// TIA Portal project "vfd-spindel-plc_v20" (V20)

(* hardware
DEVICE "ET 200SP station_1"  ET 200SP-Station
   slot 0: "Rack_0"  Rack  6ES5 710-8MAx1
   slot 1: "vfd-spindel-plc"  CPU 1510SP-1 PN  6ES7 510-1DJ01-0AB0  V2.5
      slot 32768: "PROFINET interface_1"  X1
         slot 32771: "Port_3"  X1 P3
   slot 2: "AQ 4xU/I ST_1"  AQ 4xU/I ST  6ES7 135-6HD00-0BA1  V1.1
      slot 1: "AQ 4xU/I ST_1"  AQ 4xU/I ST
   slot 3: "AI 2xU/I 2-/4-wire HS_1"  AI 2xU/I 2-,4-wire HS  6ES7 134-6HB00-0DA1  V2.0
      slot 1: "AI 2xU/I 2-/4-wire HS_1"  AI 2xU/I 2-,4-wire HS
   slot 4: "DQ 8x24VDC/0.5A HF_1"  DQ 8x24VDC/0.5A HF  6ES7 132-6BF00-0CA0  V2.0
      slot 1: "DQ 8x24VDC/0.5A HF_1"  DQ 8x24VDC/0.5A HF
   slot 5: "DQ 8x24VDC/0.5A HF_2"  DQ 8x24VDC/0.5A HF  6ES7 132-6BF00-0CA0  V2.0
      slot 1: "DQ 8x24VDC/0.5A HF_2"  DQ 8x24VDC/0.5A HF
   slot 6: "DI 8x24VDC HF_1"  DI 8x24VDC HF  6ES7 131-6BF00-0CA0  V2.0
      slot 1: "DI 8x24VDC HF_1"  DI 8x24VDC HF
   slot 7: "TM Count 1x24V_1"  TM Count 1x24V  6ES7 138-6AA01-0BA0  V2.0
      slot 1: "TM Count 1x24V_1"  TM Count 1x24V
   slot 8: "AI 4xRTD/TC 2-/3-/4-wire HF_1"  AI 4xRTD/TC 2-,3-,4-wire HF  6ES7 134-6JD00-0CA1  V2.0
      slot 1: "AI 4xRTD/TC 2-/3-/4-wire HF_1"  AI 4xRTD/TC 2-,3-,4-wire HF
   slot 9: "Server module_1"  Server module  6ES7 193-6PA00-0AA0  V1.1
      slot 1: "Server module_1"  Server module
   slot 127: "BA 2xRJ45"  BA 2xRJ45  6ES7 193-6AR00-0AA0  V0.0
      slot 32769: "Port_1"  X1 P1  6ES7 193-6AR00-0AA0
      slot 32770: "Port_2"  X1 P2  6ES7 193-6AR00-0AA0
DEVICE "ktp700_basic"  KTP700 Basic PN
   slot 0: "ktp700_basic"  KTP700 Basic PN  6AV2 123-2GB03-0AX0  17.0.0.0
   slot 1: "HMI_RT_1"  KTP700 Basic PN  6AV2 123-2GB03-0AX0  17.0.0.0
   slot 5: "ktp700_basic.IE_CP_1"  PROFINET Interface  17.0.0.0
      slot 1: "PROFINET Interface_1"  PROFINET Interface
         slot 1: "Port_1"  Port
*)

// ===== PLC "vfd-spindel-plc"  CPU 1510SP-1 PN =====

VAR_GLOBAL   // PLC tag table "Default tag table"
   "DQ0" AT %Q8.0 : Bool;
   "AQ_Ch1" AT %QW0 : Word;
   "AI_Ch0" AT %IW0 : Word;
   "AQ_Ch2" AT %QW2 : Word;
   "AI_Ch1" AT %IW2 : Word;
   "AQ_Ch3" AT %QW4 : Word;
   "AQ_Ch4" AT %QW6 : Word;
   "DI4" AT %I28.3 : Bool;   // Safety relay
   "DI5" AT %I28.4 : Bool;   // Safety button
   "AI1_RTD" AT %IW6 : Word;
   "AI2_RTD" AT %IW8 : Word;
   "DI0_safetyRelay" AT %I28.0 : Bool;
   "DQ1" AT %Q8.1 : Bool;
   "DQ4" AT %Q8.4 : Bool;
   "DI1_SafetyRelay_State" AT %I28.1 : Bool;
END_VAR

TYPE "UDT_IO_AI"
   STRUCT
      AI1_TeplotaKomaraKartac_Ohm : Int;
   END_STRUCT;
END_TYPE

TYPE "UDT_IO_AQ"
   STRUCT
      SpeedVoltage : Real;
      AQ2_VoltageCtrl_V : Real;
      AQ3_CurrentCtrl_V : Real;
   END_STRUCT;
END_TYPE

TYPE "UDT_IO_DI"
   STRUCT
      SafetyRelayAuxOk : Bool;
      HSC_Couter : UInt;
      EmergencyStop : Bool;
      ExternalFault : Bool;
   END_STRUCT;
END_TYPE

TYPE "UDT_IO_DQ"
   STRUCT
      EmergencyStop : Bool;
      RunForwardCmd : Bool;
      FaultResetCmd : Bool;
      MultiSpeed1 : Bool;
      ExternalFault : Bool;
      DO_OutputOff : Bool;
   END_STRUCT;
END_TYPE

TYPE "UDT_LABPSU_STATUS"
   STRUCT
      VoltageSet_V : Real;
      CurrentSet_A : Real;
      State : USInt;
      StatusText : String[40];
   END_STRUCT;
END_TYPE

TYPE "UDT_SPINDEL_STATUS"
   STRUCT
      RunLatched : Bool;
      TripActive : Bool;
      State : USInt;
      StatusText : String[40];
   END_STRUCT;
END_TYPE

TYPE "UDT_SAFETY_STATUS"
   STRUCT
      SafetyOk : Bool;
      PermitMotion : Bool;
      TripActive : Bool;
      TripCode : USInt;
      StatusText : String[40];
   END_STRUCT;
END_TYPE

DATA_BLOCK "DAC"   // DB2
{ S7_Optimized_Access := 'TRUE' }
VERSION : 0.1
   VAR
      IccLimiter : Struct
         MaxOutputCurrent : Int := 60;
         MinOutputCurrent : Int := 0;
         MinDacRange : Int := 0;
         MaxDacRange : Int := 27648;
         value : UInt := 0;
      END_STRUCT;
      UccVoltage : Struct
         MaxOutput : Int := 10;
         MinOutput : Int := 0;
         MinDacRange : Int := 0;
         MaxDacRange : Int := 27648;
      END_STRUCT;
      VFD : Struct
         MaxFrequency : Int := 18000;
         MinFrequency : Int := 0;
         MinDacRange : Int := 0;
         value : UInt := 0;
         MaxDacRange : Int := 27648;
      END_STRUCT;
      Sinus : Struct
         Value : Real := 0.0;
         Sample : Int := 0;
         Amplitude : Real := 1.0;
         Period : Real := 1.0;
         SamplePeriod : Real := 0.01;
      END_STRUCT;
   END_VAR
BEGIN
END_DATA_BLOCK

DATA_BLOCK "SpindelControl"   // DB3
{ S7_Optimized_Access := 'TRUE' }
VERSION : 0.1
   VAR
      RunForward : Bool := false;
      EmergencyStop : Bool := false;
      FaultReset : Bool := false;
      MultiSpeed1 : Bool := false;
      ExternelFault : Bool := false;
      CurrentLimiter : Real := 0.0;
      SupplyVoltage : Real := 0.0;
   END_VAR
BEGIN
END_DATA_BLOCK

DATA_BLOCK "DB_IO"   // DB4
{ S7_Optimized_Access := 'TRUE' }
VERSION : 0.1
   VAR
      DQ : "UDT_IO_DQ";
      DI : "UDT_IO_DI";
      AI : "UDT_IO_AI";
      AQ : "UDT_IO_AQ";
   END_VAR
BEGIN
END_DATA_BLOCK

DATA_BLOCK "Spindel"   // DB5
{ S7_Optimized_Access := 'TRUE' }
VERSION : 0.1
// stored: InstanceOfName FB_DriveCtrl
"FB_DriveCtrl"
BEGIN
END_DATA_BLOCK

DATA_BLOCK "DB_Status"   // DB6
{ S7_Optimized_Access := 'TRUE' }
VERSION : 0.1
   VAR
      Spindel : "UDT_SPINDEL_STATUS";
      Safety : "UDT_SAFETY_STATUS";
      LabPSU : "UDT_LABPSU_STATUS";
   END_VAR
BEGIN
END_DATA_BLOCK

DATA_BLOCK "LabPSU"   // DB7
{ S7_Optimized_Access := 'TRUE' }
VERSION : 0.1
// stored: InstanceOfName FB_LabPSU
"FB_LabPSU"
BEGIN
END_DATA_BLOCK

DATA_BLOCK "LabPSU_Control"   // DB8
{ S7_Optimized_Access := 'TRUE' }
VERSION : 0.1
   VAR
      Enable : Bool := false;
      PermitOutput : Bool := false;
      Mode : USInt := 0;
      Cycle_s : Real := 0.01;
      BaseVoltage_V : Real := 1.0;
      CurrentOffset_A : Real := 0.0;
      DebugAmplitude_A : Real := 60.0;
      DebugFrequency_Hz : Real := 2.0;
      ConstCurrent_A : Real := 10.0;
   END_VAR
BEGIN
END_DATA_BLOCK

DATA_BLOCK "Safety_1"   // DB9
{ S7_Optimized_Access := 'TRUE' }
VERSION : 0.1
// stored: InstanceOfName FB_SafetyGate
"FB_SafetyGate"
BEGIN
END_DATA_BLOCK

DATA_BLOCK "DB_Alarms"   // DB10
{ S7_Optimized_Access := 'TRUE' }
VERSION : 0.1
   VAR
      TempHigh : Bool;
      VibCritical : Bool;
   END_VAR
BEGIN
END_DATA_BLOCK

DATA_BLOCK "DB_HMI"   // DB11
{ S7_Optimized_Access := 'TRUE' }
VERSION : 0.1
   VAR
      System : Struct
         Enable : Bool;
      END_STRUCT;
      Spindle : Struct
         Start : Bool;
         Stop : Bool;
         ResetFault : Bool;
         Speed_RPM : Real;
         Enable : Bool;
      END_STRUCT;
      LabPSU : Struct
         Enable : Bool;
         Mode : Bool;
         BaseVoltage_V : Bool;
         DebugAmplitude_A : Bool;
         DebugFrequency_Hz : Bool;
         CurrentOffset_A : Bool;
         ConstCurrent_A : Bool;
      END_STRUCT;
   END_VAR
BEGIN
END_DATA_BLOCK

FUNCTION_BLOCK "FB_DriveCtrl"   // FB1, SCL
{ S7_Optimized_Access := 'TRUE' }
VERSION : 0.1
   VAR_INPUT
      HMI_Start : Bool := false;   // start command (button)
      HMI_Stop : Bool := false;   // stop command (button)
      HMI_ResetFault : Bool := false;   // reset fault (button)
      HMI_Speed_RPM : Real := 0.0;   // speed setpoint in RPM Interlocks / safety
      PermitMotion : Bool := false;   // from safety gate
      EmergencyStop : Bool := false;   // E-Stop chain
      ExternalFaultIn : Bool := false;   // external fault input Parameters
      SpeedMax_RPM : Real := 18000.0;   // max RPM corresponds to 10V
      AO_MaxVolt : Real := 10.0;   // 0..10V
      RampUp_RPM_per_s : Real := 6000.0;   // ramp up rate
      RampDown_RPM_per_s : Real := 9000.0;   // ramp down rate
      ResetPulse : Time := T#300MS;   // reset pulse length
      RequireSpeedToRun : Bool := FALSE;   // if TRUE, Start only latches when setpoint > 0 Outputs to drive
   END_VAR
   VAR_OUTPUT
      DO_RunForward : Bool := false;
      DO_FaultReset : Bool := false;
      DO_MultiSpeed1 : Bool := false;
      DO_ExternalFault : Bool := false;
      AQ1_Voltage_0_10V : Real := 0.0;   // Status for HMI/diagnostics
      RunLatched : Bool := false;   // internal run request latch
      TripActive : Bool := false;   // interlock active
      State : USInt := 0;   // 0 STOPPED, 1 RUN_CMD, 2 STOPPING, 3 TRIP
      StatusText : String[40] := '';   // Edge detection
   END_VAR
   VAR
      prevStart : Bool := false;
      prevStop : Bool := false;
      prevReset : Bool := false;
      startEdge : Bool := false;
      stopEdge : Bool := false;
      resetEdge : Bool := false;   // Ramp variables
      speedCmdRPM : Real := 0.0;
      speedRampRPM : Real := 0.0;   // Reset pulse timer
      tReset : TON_TIME;   // Cycle time assumption (OB1). Use OB35 for precise timing if needed.
      cycle_s : Real := 0.01;   // 10 ms default
   END_VAR
BEGIN
       // ------------------------------------------------------------
       // Edge detection for Start/Stop/Reset
       // ------------------------------------------------------------
       #startEdge := #HMI_Start AND NOT #prevStart;
       #stopEdge := #HMI_Stop AND NOT #prevStop;
       #resetEdge := #HMI_ResetFault AND NOT #prevReset;

       #prevStart := #HMI_Start;
       #prevStop := #HMI_Stop;
       #prevReset := #HMI_ResetFault;

       // ------------------------------------------------------------
       // Trip / interlock
       // Trip znamena zakaz běhu vřetene, pokud není splněna bezpečnostní podmínka. Trip = okamžité odstavení zařízení.
       // ------------------------------------------------------------
       #TripActive := (NOT #PermitMotion) OR #EmergencyStop OR #ExternalFaultIn;

       // External fault output to the drive (if wired this way)
       #DO_ExternalFault := #TripActive;

       // ------------------------------------------------------------
       // Sanitize setpoint
       // Sanitize = zkontrolovat a upravit vstupní hodnotu tak, aby byla bezpečná a platná.
       // ------------------------------------------------------------
       #speedCmdRPM := #HMI_Speed_RPM;
       IF #speedCmdRPM < 0.0 THEN
           #speedCmdRPM := 0.0;
       END_IF;
       IF #speedCmdRPM > #SpeedMax_RPM THEN
           #speedCmdRPM := #SpeedMax_RPM;
       END_IF;

       // ------------------------------------------------------------
       // Run latch logic (Stop has priority)
       // ------------------------------------------------------------
       IF #TripActive THEN
           #RunLatched := FALSE;
       ELSE
           IF #stopEdge OR #HMI_Stop THEN
               #RunLatched := FALSE;
           ELSIF #startEdge OR #HMI_Start THEN
               IF (NOT #RequireSpeedToRun) OR (#speedCmdRPM > 0.0) THEN
                   #RunLatched := TRUE;
               END_IF;
           END_IF;
       END_IF;

       // ------------------------------------------------------------
       // Fault reset pulse (recommended only when not running)
       // ------------------------------------------------------------
       #tReset(IN := (#resetEdge AND NOT #TripActive AND NOT #RunLatched),
               PT := #ResetPulse);
       #DO_FaultReset := #tReset.Q;

       // ------------------------------------------------------------
       // Defaults
       // ------------------------------------------------------------
       #DO_MultiSpeed1 := FALSE;

       // ------------------------------------------------------------
       // State (for HMI readability; no drive feedback available)
       // ------------------------------------------------------------
       IF #TripActive THEN
           #State := 3; // TRIP
       ELSE
           IF #RunLatched THEN
               #State := 1; // RUN_CMD
           ELSE
               IF #speedRampRPM > 0.0 THEN
                   #State := 2; // STOPPING (ramp down)
               ELSE
                   #State := 0; // STOPPED
               END_IF;
           END_IF;
       END_IF;

       CASE #State OF
           0:
               #StatusText := 'STOPPED';
           1:
               #StatusText := 'RUN CMD (no feedback)';
           2:
               #StatusText := 'STOPPING (ramp down)';
           3:
               #StatusText := 'TRIP (E-Stop/Interlock)';
           ELSE
               #StatusText := 'UNKNOWN';
       END_CASE;

       // ------------------------------------------------------------
       // Drive command + speed ramp
       // ------------------------------------------------------------
       IF #TripActive THEN
           #DO_RunForward := FALSE;
           #speedRampRPM := 0.0;
       ELSE
           IF #RunLatched THEN
               #DO_RunForward := TRUE;

               // Ramp toward setpoint (up & down)
               IF #speedRampRPM < #speedCmdRPM THEN
                   #speedRampRPM := #speedRampRPM + (#RampUp_RPM_per_s * #cycle_s);
                   IF #speedRampRPM > #speedCmdRPM THEN
                       #speedRampRPM := #speedCmdRPM;
                   END_IF;
               ELSIF #speedRampRPM > #speedCmdRPM THEN
                   #speedRampRPM := #speedRampRPM - (#RampDown_RPM_per_s * #cycle_s);
                   IF #speedRampRPM < #speedCmdRPM THEN
                       #speedRampRPM := #speedCmdRPM;
                   END_IF;
               END_IF;

           ELSE
               #DO_RunForward := FALSE;

               // Ramp down to 0
               IF #speedRampRPM > 0.0 THEN
                   #speedRampRPM := #speedRampRPM - (#RampDown_RPM_per_s * #cycle_s);
                   IF #speedRampRPM < 0.0 THEN
                       #speedRampRPM := 0.0;
                   END_IF;
               END_IF;
           END_IF;
       END_IF;

       // ------------------------------------------------------------
       // RPM -> 0..10V conversion
       // ------------------------------------------------------------
       IF #SpeedMax_RPM > 0.0 THEN
           #AQ1_Voltage_0_10V := (#speedRampRPM / #SpeedMax_RPM) * #AO_MaxVolt;
       ELSE
           #AQ1_Voltage_0_10V := 0.0;
       END_IF;

       // ------------------------------------------------------------
       // Clamp AO (Clamp znamena omezit hodnotu tak, aby zůstala v daném rozsahu (min–max))
       //  ------------------------------------------------------------
       IF #AQ1_Voltage_0_10V < 0.0 THEN
           #AQ1_Voltage_0_10V := 0.0;
       END_IF;
       IF #AQ1_Voltage_0_10V > #AO_MaxVolt THEN
           #AQ1_Voltage_0_10V := #AO_MaxVolt;
       END_IF;

       // Hard safety
       IF #TripActive THEN
           #AQ1_Voltage_0_10V := 0.0;
       END_IF;
END_FUNCTION_BLOCK

FUNCTION_BLOCK "FB_LabPSU"   // FB2, SCL
{ S7_Optimized_Access := 'TRUE' }
VERSION : 0.1
   VAR_INPUT
      Enable : Bool := false;   // povolenÃ­ funkce z PLC/HMI
      PermitOutput : Bool := false;   // interlock / safety gate
      Mode : USInt := 0;   // 0=OFF, 1=CONST, 2=SINE_DEBUG ÄasovÃ¡ zÃ¡kladna
      Cycle_s : Real := 0.01;   // typicky OB35 = 10 ms zdroj - zÃ¡kladnÃ­ nastavenÃ­
      BaseVoltage_V : Real := 1.0;   // AQ2
      CurrentOffset_A : Real := 0.0;   // DC offset proudu
      DebugAmplitude_A : Real := 60.0;   // amplituda sinu pro debug
      DebugFrequency_Hz : Real := 2.0;   // frekvence sinu pro debug konstantnÃ­ reÅ¾im
      ConstCurrent_A : Real := 10.0;   // rampy
      RampUp_A_per_s : Real := 50.0;
      RampDown_A_per_s : Real := 80.0;   // parametry zdroje BK1900B
      PSU_MaxVoltage_V : Real := 16.0;   // model 1900B
      PSU_MaxCurrent_A : Real := 60.0;   // model 1900B
      RemoteMaxCtrl_V : Real := 5.0;   // analog remote 0..5 V engineering outputs
   END_VAR
   VAR_OUTPUT
      VoltageSet_V : Real := 0.0;   // poÅ¾adovanÃ© napÄ›tÃ­ zdroje
      CurrentSet_A : Real := 0.0;   // poÅ¾adovanÃ½ current limit analog outputs for PLC IO layer
      AQ2_VoltageCtrl_V : Real := 0.0;   // 0..5 V na pin 2
      AQ3_CurrentCtrl_V : Real := 0.0;   // 0..5 V na pin 3 digital output for pin 5
      DO_OutputOff : Bool := false;   // TRUE = vypnout vÃ½stup zdroje status
      State : USInt := 0;   // 0 OFF, 1 CONST, 2 SINE
      StatusText : String[40] := '';
   END_VAR
   VAR
      phase_rad : Real := 0.0;
      omega : Real := 0.0;
      targetCurrent_A : Real := 0.0;
      sineValue : Real := 0.0;
   END_VAR
BEGIN
       // default
       #VoltageSet_V := 0.0;
       #CurrentSet_A := 0.0;
       #AQ2_VoltageCtrl_V := 0.0;
       #AQ3_CurrentCtrl_V := 0.0;
       #DO_OutputOff := TRUE;
       #State := 0;
       #StatusText := 'OFF';

       // safety / permit
       IF (NOT #Enable) OR (NOT #PermitOutput) THEN
           #phase_rad := 0.0;
           RETURN;
       END_IF;

       // vÃ½stup zdroje povolen
       #DO_OutputOff := FALSE;

       // zÃ¡kladnÃ­ napÄ›tÃ­
       #VoltageSet_V := #BaseVoltage_V;

       // omezenÃ­ napÄ›tÃ­
       IF #VoltageSet_V < 0.0 THEN
           #VoltageSet_V := 0.0;
       END_IF;
       IF #VoltageSet_V > #PSU_MaxVoltage_V THEN
           #VoltageSet_V := #PSU_MaxVoltage_V;
       END_IF;

       CASE #Mode OF
           0: // OFF
               #CurrentSet_A := 0.0;
               #State := 0;
               #StatusText := 'OFF';

           1: // CONST
               #targetCurrent_A := #ConstCurrent_A;

               IF #targetCurrent_A < 0.0 THEN
                   #targetCurrent_A := 0.0;
               END_IF;
               IF #targetCurrent_A > #PSU_MaxCurrent_A THEN
                   #targetCurrent_A := #PSU_MaxCurrent_A;
               END_IF;

               // jednoduchÃ¡ rampa
               IF #CurrentSet_A < #targetCurrent_A THEN
                   #CurrentSet_A := #CurrentSet_A + (#RampUp_A_per_s * #Cycle_s);
                   IF #CurrentSet_A > #targetCurrent_A THEN
                       #CurrentSet_A := #targetCurrent_A;
                   END_IF;
               ELSIF #CurrentSet_A > #targetCurrent_A THEN
                   #CurrentSet_A := #CurrentSet_A - (#RampDown_A_per_s * #Cycle_s);
                   IF #CurrentSet_A < #targetCurrent_A THEN
                       #CurrentSet_A := #targetCurrent_A;
                   END_IF;
               END_IF;

               #State := 1;
               #StatusText := 'CONST';

           2: // SINE_DEBUG
               #omega := 6.2831853 * #DebugFrequency_Hz; // 2*pi*f

               #phase_rad := #phase_rad + (#omega * #Cycle_s);

               // drÅ¾et fÃ¡zi v rozumnÃ©m rozsahu
               IF #phase_rad > 6.2831853 THEN
                   #phase_rad := #phase_rad - 6.2831853;
               END_IF;

               #sineValue := SIN(#phase_rad);

               // sinus s offsetem
               #targetCurrent_A := #CurrentOffset_A + (#DebugAmplitude_A * #sineValue);

               // current limit zdroje nemÅ¯Å¾e bÃ½t zÃ¡pornÃ½
               IF #targetCurrent_A < 0.0 THEN
                   #targetCurrent_A := 0.0;
               END_IF;
               IF #targetCurrent_A > #PSU_MaxCurrent_A THEN
                   #targetCurrent_A := #PSU_MaxCurrent_A;
               END_IF;

               // volitelnÄ› mÅ¯Å¾eÅ¡ i tady nechat rampu, ale pro sinus ji vÄ›tÅ¡inou nechceÅ¡ moc agresivnÃ­
               #CurrentSet_A := #targetCurrent_A;

               #State := 2;
               #StatusText := 'SINE DEBUG';

           ELSE
               #CurrentSet_A := 0.0;
               #State := 0;
               #StatusText := 'UNKNOWN->OFF';
       END_CASE;

       // pÅ™evod engineering units -> BK remote control 0..5V

       // napÄ›tÃ­
       IF #PSU_MaxVoltage_V > 0.0 THEN
           #AQ2_VoltageCtrl_V := (#VoltageSet_V / #PSU_MaxVoltage_V) * #RemoteMaxCtrl_V;
       ELSE
           #AQ2_VoltageCtrl_V := 0.0;
       END_IF;

       // proud
       IF #PSU_MaxCurrent_A > 0.0 THEN
           #AQ3_CurrentCtrl_V := (#CurrentSet_A / #PSU_MaxCurrent_A) * #RemoteMaxCtrl_V;
       ELSE
           #AQ3_CurrentCtrl_V := 0.0;
       END_IF;

       // clamp
       IF #AQ2_VoltageCtrl_V < 0.0 THEN
           #AQ2_VoltageCtrl_V := 0.0;
       END_IF;
       IF #AQ2_VoltageCtrl_V > #RemoteMaxCtrl_V THEN
           #AQ2_VoltageCtrl_V := #RemoteMaxCtrl_V;
       END_IF;

       IF #AQ3_CurrentCtrl_V < 0.0 THEN
           #AQ3_CurrentCtrl_V := 0.0;
       END_IF;
       IF #AQ3_CurrentCtrl_V > #RemoteMaxCtrl_V THEN
           #AQ3_CurrentCtrl_V := #RemoteMaxCtrl_V;
       END_IF;
END_FUNCTION_BLOCK

FUNCTION_BLOCK "FB_SafetyGate"   // FB3, SCL
{ S7_Optimized_Access := 'TRUE' }
VERSION : 0.1
   VAR_INPUT
      Enable : Bool;   // hlavní povolení systému
      EmergencyStop : Bool;   // 1 = E-Stop aktivní
      SafetyRelayAuxOk : Bool;   // 1 = safety relé OK
      ExternalFault : Bool;   // 1 = externí chyba
      TempAlarm : Bool;   // 1 = kritická teplota
      VibAlarm : Bool;   // 1 = kritické vibrace
   END_VAR
   VAR_OUTPUT
      SafetyOk : Bool;
      PermitMotion : Bool;
      TripActive : Bool;
      TripCode : USInt;
      StatusText : String[40];
   END_VAR
BEGIN
   // hardware safety stav
   #SafetyOk := #SafetyRelayAuxOk AND NOT #EmergencyStop;

   // centrální trip
   #TripActive := (NOT #SafetyOk)OR #ExternalFault OR #TempAlarm OR #VibAlarm OR (NOT #Enable);

   // povolení pohybu
   #PermitMotion := NOT #TripActive;

   // diagnostika
   IF #EmergencyStop THEN
       #TripCode := 1;
       #StatusText := 'E-STOP ACTIVE';
   ELSIF NOT #SafetyRelayAuxOk THEN
       #TripCode := 2;
       #StatusText := 'SAFETY RELAY NOT OK';
   ELSIF #ExternalFault THEN
       #TripCode := 3;
       #StatusText := 'EXTERNAL FAULT';
   ELSIF #TempAlarm THEN
       #TripCode := 4;
       #StatusText := 'TEMP ALARM';
   ELSIF #VibAlarm THEN
       #TripCode := 5;
       #StatusText := 'VIBRATION ALARM';
   ELSIF NOT #Enable THEN
       #TripCode := 6;
       #StatusText := 'SYSTEM NOT ENABLED';
   ELSE
       #TripCode := 0;
       #StatusText := 'READY';
   END_IF;
END_FUNCTION_BLOCK

FUNCTION "FC_Scale" : Real   // FC2, SCL
{ S7_Optimized_Access := 'TRUE' }
VERSION : 0.1
   VAR_INPUT
      InValue : Real;   // vstupní hodnota (engineering units), napr. napeti pro DA prevodnik pro ovladani otacek
      InMin : Real;   // minimum vstupního rozsahu, ie 0.0V
      InMax : Real;   // maximum vstupního rozsahu, ie 10.0V
      OutMin : Real;   // minimum výstupního rozsahu, ie. 0.0 (minimalni hodnota prevodniku)
      OutMax : Real;   // maximum výstupního rozsahu, ie. 27648.0 (maximalni hodnota DA prevodniku)
   END_VAR
   VAR_TEMP
      Ratio : Real;
   END_VAR
BEGIN
   // ochrana proti dělení nulou
   IF (#InMax - #InMin) = 0.0 THEN
       #FC_Scale := #OutMin;
       RETURN;
   END_IF;

   // normalizace vstupu (0..1)
   #Ratio := (#InValue - #InMin) / (#InMax - #InMin);

   // škálování do výstupního rozsahu
   #FC_Scale := #OutMin + #Ratio * (#OutMax - #OutMin);
END_FUNCTION

FUNCTION "FC_IO_Map_Write" : Void   // FC3, SCL
{ S7_Optimized_Access := 'TRUE' }
VERSION : 0.1
BEGIN
   //ZAPIS NA VYSTUPY
   // AQ1+, AQ1-  [Měnič] AVI, ACM
   // AQ2+, AQ2-  [Labor. zdroj] U_LabPSU Nastavení výstupního napětí na svorkách laboratorního zdroje. Napětí by mělo jít vypočítat proud a odpor na uhlíku.
   // AQ3+, AQ3-  [Labor. zdroj] I_LabPSU Řízení proudové ochrany laboratorního zdroje., neboli ovládání frekvence a amplitudy

   "AQ_Ch1" := REAL_TO_INT("FC_Scale"(InMin := 0.0, InMax := 10.0, InValue := "DB_IO".AQ.SpeedVoltage, OutMin := 0.0, OutMax := "DAC".VFD.MaxDacRange));
   "AQ_Ch2" := REAL_TO_INT("DB_IO".AQ.AQ2_VoltageCtrl_V / 10.0 * 27648.0);
   "AQ_Ch3" := REAL_TO_INT("DB_IO".AQ.AQ3_CurrentCtrl_V / 10.0 * 27648.0);

   "DQ0" := "DB_IO".DQ.RunForwardCmd;
   "DQ1" := NOT "DI0_safetyRelay";
   "DQ4" := NOT "DI1_SafetyRelay_State";
END_FUNCTION

FUNCTION "FC_IO_Map_Read" : Void   // FC4, SCL
{ S7_Optimized_Access := 'TRUE' }
VERSION : 0.1
BEGIN
   //"DB_IO".DI.SafetyRelayAuxOk := "DI0_safetyRelay";
   "DB_IO".DI.EmergencyStop := "DI5";
   "DB_IO".AI.AI1_TeplotaKomaraKartac_Ohm := "AI1_RTD";
END_FUNCTION

ORGANIZATION_BLOCK "Main"   // OB1, SCL, ProgramCycle
TITLE = "Main Program Sweep (Cycle)"
{ S7_Optimized_Access := 'TRUE' }
VERSION : 0.1
   VAR_INPUT
      Initial_Call : Bool;   // Initial call of this OB
      Remanence : Bool;   // =True, if remanent data are available
   END_VAR
   VAR_TEMP
      WwwRetVal : Int;
   END_VAR
BEGIN
   //******************************************************************
   //ESTABLISH WEBSERVER
   #WwwRetVal := WWW("DB 333");
   //******************************************************************

   //******************************************************************
   // IO MAP READ
   //******************************************************************
   "FC_IO_Map_Read"();

   //******************************************************************
   // CALL FB BLOCKS - PRODUCTION LOGIC
   //******************************************************************
   //Nektere safety signaly nemame implementovane - teplota, vibrace. Zatim bude potreba je simulovat
   "Safety_1"(Enable:= TRUE, // This signal can be used to bind to another system in the future 
              EmergencyStop:="DB_IO".DI.EmergencyStop,
              SafetyRelayAuxOk:= "DB_IO".DI.SafetyRelayAuxOk,
              ExternalFault:= "DB_IO".DI.ExternalFault,
              TempAlarm:="DB_Alarms".TempHigh,
              VibAlarm:= "DB_Alarms".VibCritical,
              SafetyOk => "DB_Status".Safety.SafetyOk,
              PermitMotion => "DB_Status".Safety.PermitMotion,
              TripActive => "DB_Status".Safety.TripActive,
              TripCode => "DB_Status".Safety.TripCode,
              StatusText => "DB_Status".Safety.StatusText
   );


   "Spindel"(HMI_Start:= "DB_HMI".Spindle.Start,
             HMI_Stop:="DB_HMI".Spindle.Stop,
             HMI_ResetFault:="DB_HMI".Spindle.ResetFault,
             HMI_Speed_RPM:="DB_HMI".Spindle.Speed_RPM,
             PermitMotion:="DB_Status".Safety.PermitMotion,
             EmergencyStop:="DB_IO".DI.EmergencyStop,
             ExternalFaultIn:="DB_IO".DI.ExternalFault,
             SpeedMax_RPM:=18000.0,
             AO_MaxVolt:=10.0,
             RampUp_RPM_per_s:=6000.0,
             RampDown_RPM_per_s:=9000.0,
             ResetPulse:=T#300MS,
             RequireSpeedToRun:=FALSE,
             DO_RunForward=>"DB_IO".DQ.RunForwardCmd,
             DO_FaultReset=>"DB_IO".DQ.FaultResetCmd,
             DO_MultiSpeed1=>"DB_IO".DQ.MultiSpeed1,
             DO_ExternalFault=>"DB_IO".DQ.ExternalFault,
             AQ1_Voltage_0_10V=>"DB_IO".AQ.SpeedVoltage,
             RunLatched=>"DB_Status".Spindel.RunLatched,
             TripActive=>"DB_Status".Spindel.TripActive,
             State=>"DB_Status".Spindel.State,
             StatusText=>"DB_Status".Spindel.StatusText);



   //******************************************************************
   // CALL OTHER FB BLOCKS
   //******************************************************************

   //******************************************************************
   // IO MAP WRITE
   //******************************************************************
   "FC_IO_Map_Write"();
END_ORGANIZATION_BLOCK

ORGANIZATION_BLOCK "TimeSensitive"   // OB30, SCL, CyclicInterrupt
{ S7_Optimized_Access := 'TRUE' }
VERSION : 0.1
   VAR_INPUT
      Initial_Call : Bool;   // Initial call of this OB
      Event_Count : Int;   // Events discarded
   END_VAR
   VAR_TEMP
      NormValue : Real;
      ScaledValue : UInt;
   END_VAR
   VAR CONSTANT
      PI : Real := 3.141593;
   END_VAR
BEGIN
   "LabPSU"(Enable := "LabPSU_Control".Enable,
            PermitOutput := "LabPSU_Control".PermitOutput,
            Mode := "LabPSU_Control".Mode,
            Cycle_s := "LabPSU_Control".Cycle_s,
            BaseVoltage_V := "LabPSU_Control".BaseVoltage_V,
            CurrentOffset_A := "LabPSU_Control".CurrentOffset_A,
            DebugAmplitude_A := "LabPSU_Control".DebugAmplitude_A,
            DebugFrequency_Hz := "LabPSU_Control".DebugFrequency_Hz,
            ConstCurrent_A := "LabPSU_Control".ConstCurrent_A,
            RampUp_A_per_s := 50.0,
            RampDown_A_per_s := 80.0,
            PSU_MaxVoltage_V := 16.0,
            PSU_MaxCurrent_A := 60.0,
            RemoteMaxCtrl_V := 5.0,
            VoltageSet_V => "DB_Status".LabPSU.VoltageSet_V,
            CurrentSet_A => "DB_Status".LabPSU.CurrentSet_A,
            AQ2_VoltageCtrl_V => "DB_IO".AQ.AQ2_VoltageCtrl_V,
            AQ3_CurrentCtrl_V => "DB_IO".AQ.AQ3_CurrentCtrl_V,
            DO_OutputOff => "DB_IO".DQ.DO_OutputOff,
            State => "DB_Status".LabPSU.State,
            StatusText => "DB_Status".LabPSU.StatusText);
END_ORGANIZATION_BLOCK

(* ===== HMI "HMI_RT_1" =====
system functions are stored by id; their names below are inferred from use
connection "HMI_Connection_1": ETHERNET, SMART_S7_1500_OMS

HMI tags "Default tag table"
   "Tag_ScreenNumber" : UInt, internal
   "Spindel_HMI_Start" : Bool = PLC Spindel.HMI_Start, 1 s
   "Spindel_HMI_Stop" : Bool = PLC Spindel.HMI_Stop, 1 s
   "Spindel_DO_ExternalFault" : Bool = PLC Spindel.DO_ExternalFault, 1 s
   "Spindel_HMI_Speed_RPM" : Real = PLC Spindel.HMI_Speed_RPM, 1 s
   "LabPSU_DebugAmplitude_A" : Real = PLC LabPSU.DebugAmplitude_A, 1 s
   "LabPSU_Control_DebugFrequency_Hz" : Real = PLC LabPSU_Control.DebugFrequency_Hz, 1 s
   "DB_HMI_Spindle_Start" : Bool = PLC DB_HMI.Spindle.Start, 1 s
   "DB_HMI_Spindle_Stop" : Bool = PLC DB_HMI.Spindle.Stop, 1 s
   "DB_HMI_Spindle_Speed_RPM" : Real = PLC DB_HMI.Spindle.Speed_RPM, 1 s

HMI tags "Buttons"
   "Start_activated" : Bool, internal
   "Stop_activated" : Bool, internal

graphic list "Graphic_list_1": 0 'PilotLight_Round_R_Off_256c'; 1 'PilotLight_Round_R_On_256c'

graphic list "@DiagnosticsStates": 0 '@Diagnostics_StateGood'; 1 '@Diagnostics_StateBad'

screen "Home" 800x480, template "General"
   on GenerateScreen: SetTag("Tag_ScreenNumber", 1)
   Softkey "Softkey_F2" at 0,0 size 0x0
      on KeyDown: ActivateScreen("Spindel", 0)
   Softkey "Softkey_F3" at 0,0 size 0x0
      on KeyDown: ActivateScreen("LabPSU", 0)
   TextField "Text field_6" at 65,203 size 264x34; Text 'Požadované hodnoty'
   Button "Button_1" at 21,106 size 156x82; TextOff 'START'
      on Press: SetBit("DB_HMI_Spindle_Start"); SetBit("Start_activated"); ResetBit("Stop_activated")
      Appearance <- "Start_activated"
   Button "Button_2" at 208,106 size 156x82; TextOff 'STOP'
      on Press: ResetBit("DB_HMI_Spindle_Stop"); SetBit("Stop_activated"); ResetBit("Start_activated")
      Appearance <- "Stop_activated"
   IOField "I/O field_3" at 126,253 size 170x47; FormatPattern 99999
      ProcessValue <- "DB_HMI_Spindle_Speed_RPM"
   TextField "Text field_2" at 301,262 size 59x29; Text 'RPM'
   TextField "Text field_7" at 33,262 size 79x29; Text 'Otáčky'
   IOField "I/O field_1" at 127,311 size 170x47; FormatPattern 99999
      ProcessValue <- "LabPSU_DebugAmplitude_A"
   TextField "Text field_3" at 305,320 size 19x29; Text 'A'
   TextField "Text field_8" at 34,320 size 67x29; Text 'Proud'
   TextField "Text field_1" at 408,38 size 219x34; Text 'Aktuální hodnoty'
   IOField "I/O field_2" at 493,86 size 149x37; FormatPattern 99999
   TextField "Text field_4" at 651,91 size 54x27; Text 'RPM'
   TextField "Text field_5" at 410,91 size 71x27; Text 'Otáčky'
   TextField "Text field_9" at 652,138 size 18x27; Text 'A'
   TextField "Text field_10" at 410,138 size 61x27; Text 'Proud'
   TextField "Text field_11" at 652,185 size 18x27; Text 'V'
   TextField "Text field_12" at 410,185 size 68x27; Text 'Napětí'
   TextField "Text field_13" at 650,233 size 18x27; Text 'C'
   TextField "Text field_14" at 410,226 size 73x42; Text 'Teplota vřetene'
   TextField "Text field_15" at 651,280 size 18x27; Text 'C'
   TextField "Text field_16" at 410,273 size 68x42; Text 'Teplota kartáčů'
   TextField "Text field_17" at 652,328 size 17x27; Text 'g'
   TextField "Text field_18" at 410,328 size 76x27; Text 'Vibrace'
   IOField "I/O field_4" at 494,133 size 149x37; FormatPattern 99999
   IOField "I/O field_5" at 494,180 size 149x37; FormatPattern 99999
   IOField "I/O field_6" at 492,228 size 149x37; FormatPattern 99999
   IOField "I/O field_7" at 493,275 size 149x37; FormatPattern 99999
   IOField "I/O field_8" at 493,323 size 149x37; FormatPattern 99999
   DateTimeField "Date/time field_1" at 667,9 size 116x32
   Softkey "Softkey_F1" at 0,0 size 0x0
      on KeyDown: ActivateScreen("Home", 0)

screen "LabPSU" 800x480
   Softkey "Softkey_F1" at 0,0 size 0x0
      on KeyDown: ActivateScreen("Home", 0)
   Softkey "Softkey_F3" at 0,0 size 0x0
      on KeyDown: ActivateScreen("LabPSU", 0)
   Softkey "Softkey_F2" at 0,0 size 0x0
      on KeyDown: ActivateScreen("Spindel", 0)

screen "Spindel" 800x480
   Softkey "Softkey_F2" at 0,0 size 0x0
      on KeyDown: ActivateScreen("Spindel", 0)
   Softkey "Softkey_F3" at 0,0 size 0x0
      on KeyDown: ActivateScreen("LabPSU", 0)
   Softkey "Softkey_F1" at 0,0 size 0x0
      on KeyDown: ActivateScreen("Home", 0)
*)